Fanuc KAREL source: kc00027.KL

PROGRAM KC00027
%STACKSIZE=65535
%PRIORITY=65535
%NOLOCKGROUP
VAR
I : INTEGER
J : INTEGER
K : INTEGER
R : REAL
B : BOOLEAN
S : STRING[80]
T : STRING[80]
AI : ARRAY[8] OF INTEGER
JP : JOINTPOS9
P1 : POSITION
P2 : POSITION
P3 : POSITION
AR : ARRAY[9] OF REAL
-- UNRESOLVED DECLARATIONS (source type spelling not recovered)
-- P : TYPE_0x001F (type_u16=0x001F)
-- Q : TYPE_0x001F (type_u16=0x001F)
-- AB : ARRAY[244] OF TYPE_0x0018 (type_u16=0x2018)
-- C : TYPE_0x001C (type_u16=0x001C)
BEGIN
JOINT2POS(JP,P1,P2,I,P3,C,AR,J)
END KC00027
